FUNCTION_BLOCK ABSTRACT Component IMPLEMENTS I_component
VAR
	_name : STRING;
END_VAR

METHOD ABSTRACT AddChild
VAR_INPUT
	Child : I_Component;
END_VAR
END_METHOD

METHOD FB_init : BOOL
VAR_INPUT
	bInitRetains : BOOL; // if TRUE, the retain variables are initialized (warm start / cold start)
	bInCopyCode : BOOL;  // if TRUE, the instance afterwards gets moved into the copy code (online change)
	name : STRING;
END_VAR
THIS^._name := name;
END_METHOD

METHOD ABSTRACT GetChildren : ARRAY [1..Param.NumberOfChildren] OF I_Component;
END_METHOD

PROPERTY ABSTRACT GetSize : INT
GET
END_GET
END_PROPERTY

PROPERTY Name : STRING
GET
Name := THIS^._name;
END_GET
END_PROPERTY

END_FUNCTION_BLOCK

(* stored: Version 1.1.0.1, ProductVersion 3.1.4024.12
   POU Component: Id {1ead6b77-19aa-467b-b936-a378fff952ec}, SpecialFunc None
   Folder Constructor: Id {030f87b1-3e0d-4d60-a78b-2230348806a1}
   Method AddChild: Id {a0a15808-63eb-49e1-972f-05f48a9eaa05}
   Method FB_init: Id {dc4c4cd0-6bc3-4010-84db-466007a1a384}
   Method GetChildren: Id {95f81b15-2283-488e-a4c2-996da9ff683b}
   Property GetSize: Id {5b159474-f3f4-4b12-9f7a-38cb677abfb4}
   Get Get: Id {c7251ea9-d405-4ea8-8514-fe0e6a2be71d}
   Property Name: Id {b0736d98-5438-461b-8c06-4715dbca3db8}
   Get Get: Id {ad93624a-8350-4550-8c8f-9718e37e1793} *)
